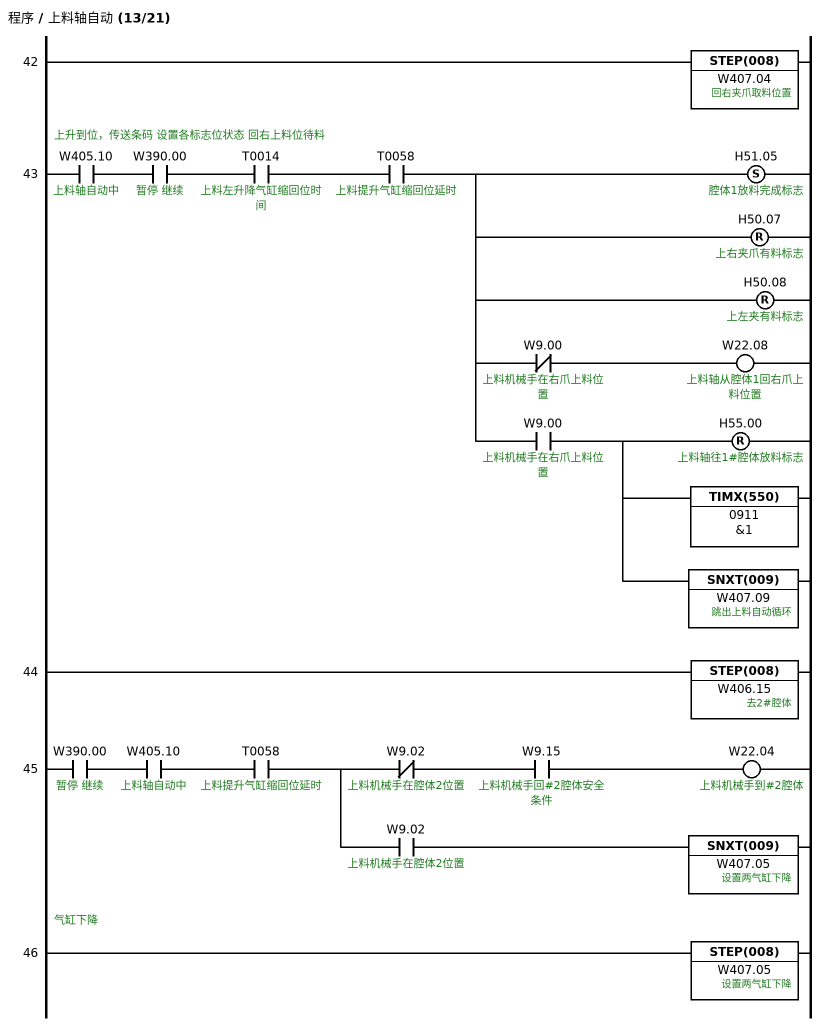
; rung 42
STEP(008) W407.04  ; 回右夹爪取料位置
; rung 43: 上升到位，传送条码 设置各标志位状态 回右上料位待料
LD W405.10  ; 上料轴自动中
AND W390.00  ; 暂停 继续
AND T0014  ; 上料左升降气缸缩回位时间
AND T0058  ; 上料提升气缸缩回位延时
OUT TR0
SET H51.05  ; 腔体1放料完成标志
RSET H50.07  ; 上右夹爪有料标志
RSET H50.08  ; 上左夹有料标志
ANDNOT W9.00  ; 上料机械手在右爪上料位置
OUT W22.08  ; 上料轴从腔体1回右爪上料位置
LD TR0
AND W9.00  ; 上料机械手在右爪上料位置
RSET H55.00  ; 上料轴往1#腔体放料标志
TIMX(550) 0911 &1
SNXT(009) W407.09  ; 跳出上料自动循环
; rung 44
STEP(008) W406.15  ; 去2#腔体
; rung 45
LD W390.00  ; 暂停 继续
AND W405.10  ; 上料轴自动中
AND T0058  ; 上料提升气缸缩回位延时
OUT TR0
ANDNOT W9.02  ; 上料机械手在腔体2位置
AND W9.15  ; 上料机械手回#2腔体安全条件
OUT W22.04  ; 上料机械手到#2腔体
LD TR0
AND W9.02  ; 上料机械手在腔体2位置
SNXT(009) W407.05  ; 设置两气缸下降
; rung 46: 气缸下降
STEP(008) W407.05  ; 设置两气缸下降

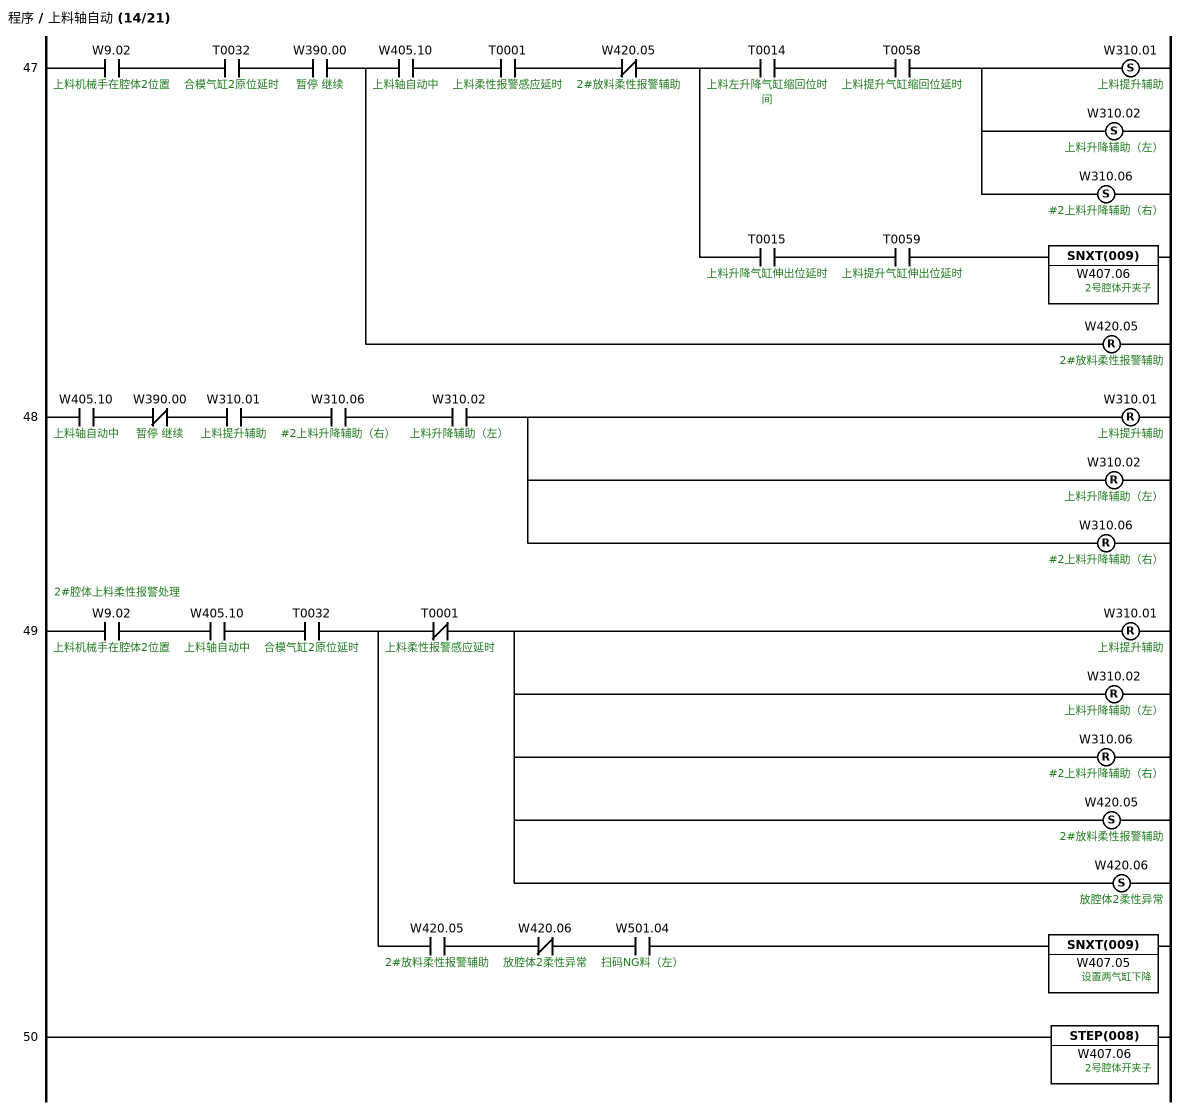
; rung 47
LD W9.02  ; 上料机械手在腔体2位置
AND T0032  ; 合模气缸2原位延时
AND W390.00  ; 暂停 继续
OUT TR0
AND W405.10  ; 上料轴自动中
AND T0001  ; 上料柔性报警感应延时
ANDNOT W420.05  ; 2#放料柔性报警辅助
OUT TR1
AND T0014  ; 上料左升降气缸缩回位时间
AND T0058  ; 上料提升气缸缩回位延时
SET W310.01  ; 上料提升辅助
SET W310.02  ; 上料升降辅助（左）
SET W310.06  ; #2上料升降辅助（右）
LD TR1
AND T0015  ; 上料升降气缸伸出位延时
AND T0059  ; 上料提升气缸伸出位延时
SNXT(009) W407.06  ; 2号腔体开夹子
LD TR0
RSET W420.05  ; 2#放料柔性报警辅助
; rung 48
LD W405.10  ; 上料轴自动中
ANDNOT W390.00  ; 暂停 继续
AND W310.01  ; 上料提升辅助
AND W310.06  ; #2上料升降辅助（右）
AND W310.02  ; 上料升降辅助（左）
RSET W310.01  ; 上料提升辅助
RSET W310.02  ; 上料升降辅助（左）
RSET W310.06  ; #2上料升降辅助（右）
; rung 49: 2#腔体上料柔性报警处理
LD W9.02  ; 上料机械手在腔体2位置
AND W405.10  ; 上料轴自动中
AND T0032  ; 合模气缸2原位延时
OUT TR0
ANDNOT T0001  ; 上料柔性报警感应延时
RSET W310.01  ; 上料提升辅助
RSET W310.02  ; 上料升降辅助（左）
RSET W310.06  ; #2上料升降辅助（右）
SET W420.05  ; 2#放料柔性报警辅助
SET W420.06  ; 放腔体2柔性异常
LD TR0
AND W420.05  ; 2#放料柔性报警辅助
ANDNOT W420.06  ; 放腔体2柔性异常
AND W501.04  ; 扫码NG料（左）
SNXT(009) W407.05  ; 设置两气缸下降
; rung 50
STEP(008) W407.06  ; 2号腔体开夹子

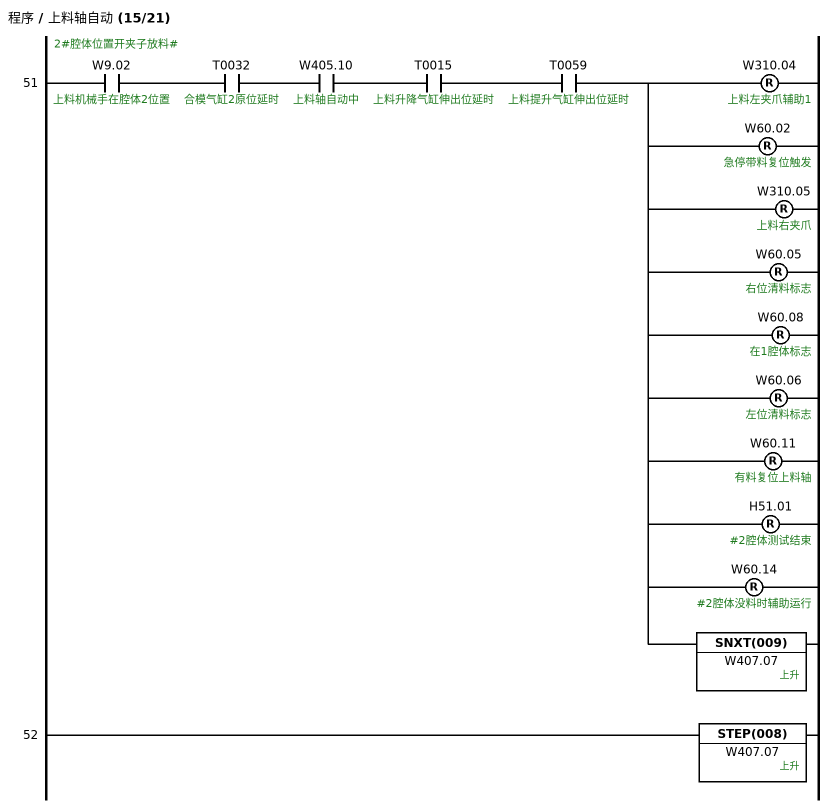
; rung 51: 2#腔体位置开夹子放料#
LD W9.02  ; 上料机械手在腔体2位置
AND T0032  ; 合模气缸2原位延时
AND W405.10  ; 上料轴自动中
AND T0015  ; 上料升降气缸伸出位延时
AND T0059  ; 上料提升气缸伸出位延时
RSET W310.04  ; 上料左夹爪辅助1
RSET W60.02  ; 急停带料复位触发
RSET W310.05  ; 上料右夹爪
RSET W60.05  ; 右位清料标志
RSET W60.08  ; 在1腔体标志
RSET W60.06  ; 左位清料标志
RSET W60.11  ; 有料复位上料轴
RSET H51.01  ; #2腔体测试结束
RSET W60.14  ; #2腔体没料时辅助运行
SNXT(009) W407.07  ; 上升
; rung 52
STEP(008) W407.07  ; 上升

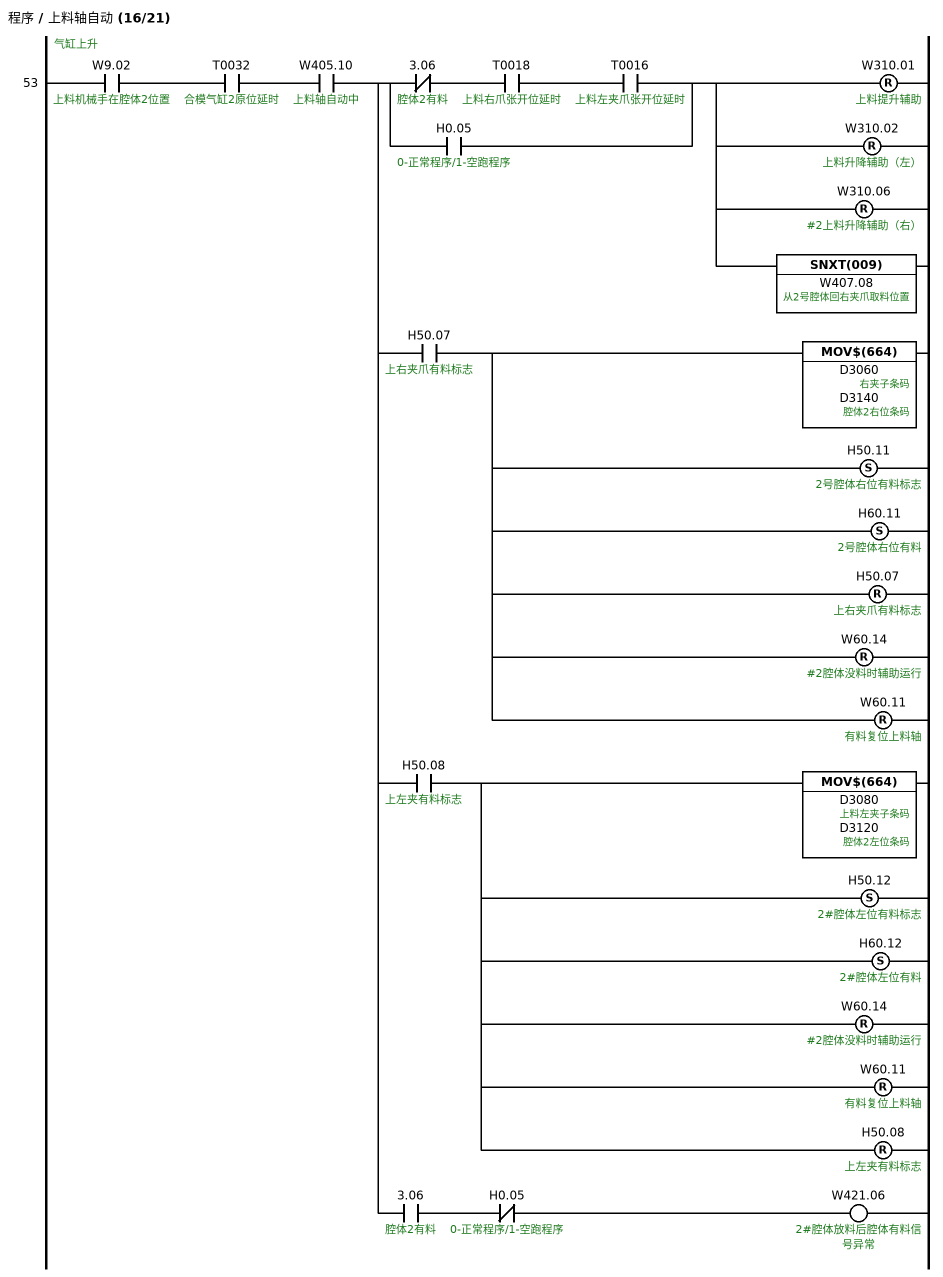
; rung 53: 气缸上升
LD W9.02  ; 上料机械手在腔体2位置
AND T0032  ; 合模气缸2原位延时
AND W405.10  ; 上料轴自动中
OUT TR0
LDNOT 3.06  ; 腔体2有料
AND T0018  ; 上料右爪张开位延时
AND T0016  ; 上料左夹爪张开位延时
OR H0.05  ; 0-正常程序/1-空跑程序
ANDLD
RSET W310.01  ; 上料提升辅助
RSET W310.02  ; 上料升降辅助（左）
RSET W310.06  ; #2上料升降辅助（右）
SNXT(009) W407.08  ; 从2号腔体回右夹爪取料位置
LD TR0
AND H50.07  ; 上右夹爪有料标志
MOV$(664) D3060 D3140  ; 右夹子条码, 腔体2右位条码
SET H50.11  ; 2号腔体右位有料标志
SET H60.11  ; 2号腔体右位有料
RSET H50.07  ; 上右夹爪有料标志
RSET W60.14  ; #2腔体没料时辅助运行
RSET W60.11  ; 有料复位上料轴
LD TR0
AND H50.08  ; 上左夹有料标志
MOV$(664) D3080 D3120  ; 上料左夹子条码, 腔体2左位条码
SET H50.12  ; 2#腔体左位有料标志
SET H60.12  ; 2#腔体左位有料
RSET W60.14  ; #2腔体没料时辅助运行
RSET W60.11  ; 有料复位上料轴
RSET H50.08  ; 上左夹有料标志
LD TR0
AND 3.06  ; 腔体2有料
ANDNOT H0.05  ; 0-正常程序/1-空跑程序
OUT W421.06  ; 2#腔体放料后腔体有料信号异常

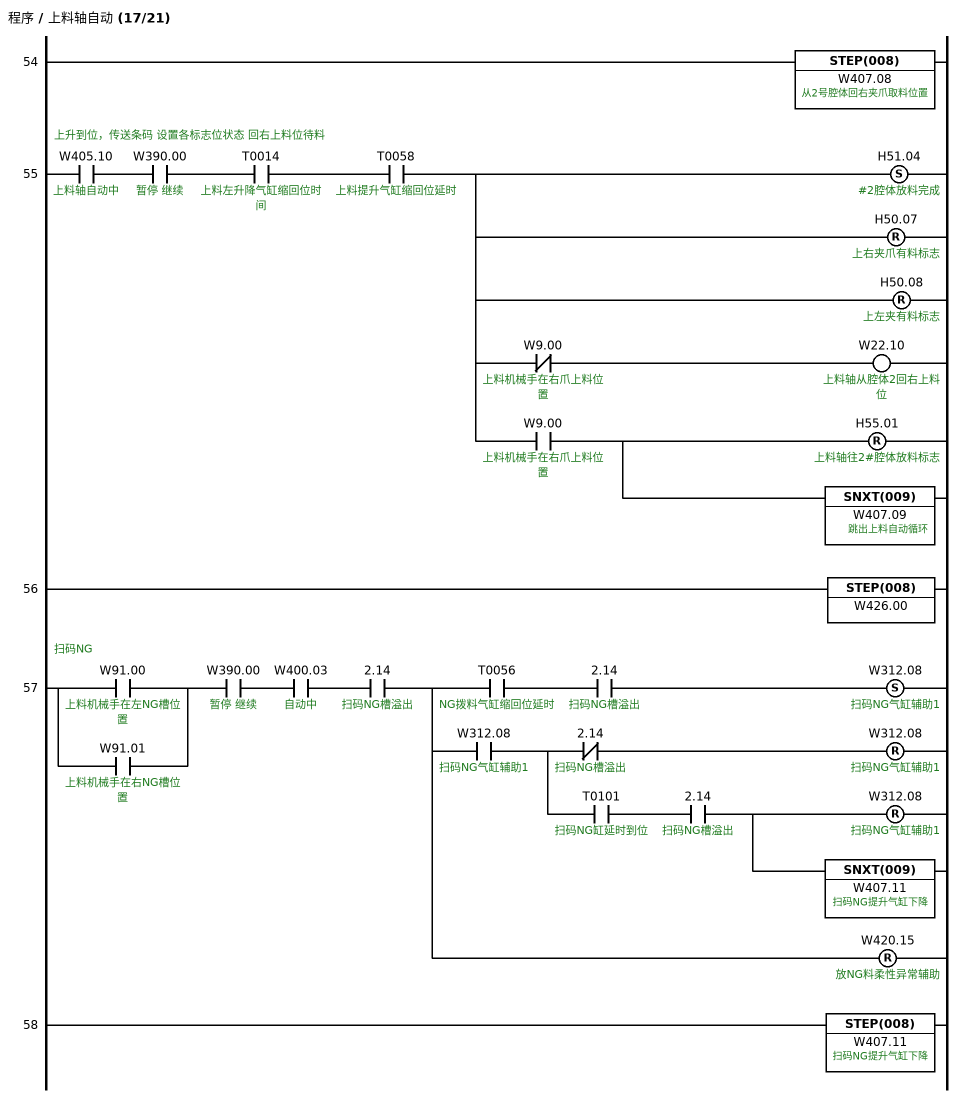
; rung 54
STEP(008) W407.08  ; 从2号腔体回右夹爪取料位置
; rung 55: 上升到位，传送条码 设置各标志位状态 回右上料位待料
LD W405.10  ; 上料轴自动中
AND W390.00  ; 暂停 继续
AND T0014  ; 上料左升降气缸缩回位时间
AND T0058  ; 上料提升气缸缩回位延时
OUT TR0
SET H51.04  ; #2腔体放料完成
RSET H50.07  ; 上右夹爪有料标志
RSET H50.08  ; 上左夹有料标志
ANDNOT W9.00  ; 上料机械手在右爪上料位置
OUT W22.10  ; 上料轴从腔体2回右上料位
LD TR0
AND W9.00  ; 上料机械手在右爪上料位置
RSET H55.01  ; 上料轴往2#腔体放料标志
SNXT(009) W407.09  ; 跳出上料自动循环
; rung 56
STEP(008) W426.00
; rung 57: 扫码NG
LD W91.00  ; 上料机械手在左NG槽位置
OR W91.01  ; 上料机械手在右NG槽位置
AND W390.00  ; 暂停 继续
AND W400.03  ; 自动中
AND 2.14  ; 扫码NG槽溢出
OUT TR0
AND T0056  ; NG拨料气缸缩回位延时
AND 2.14  ; 扫码NG槽溢出
SET W312.08  ; 扫码NG气缸辅助1
LD TR0
AND W312.08  ; 扫码NG气缸辅助1
OUT TR1
ANDNOT 2.14  ; 扫码NG槽溢出
RSET W312.08  ; 扫码NG气缸辅助1
LD TR1
AND T0101  ; 扫码NG缸延时到位
AND 2.14  ; 扫码NG槽溢出
RSET W312.08  ; 扫码NG气缸辅助1
SNXT(009) W407.11  ; 扫码NG提升气缸下降
LD TR0
RSET W420.15  ; 放NG料柔性异常辅助
; rung 58
STEP(008) W407.11  ; 扫码NG提升气缸下降

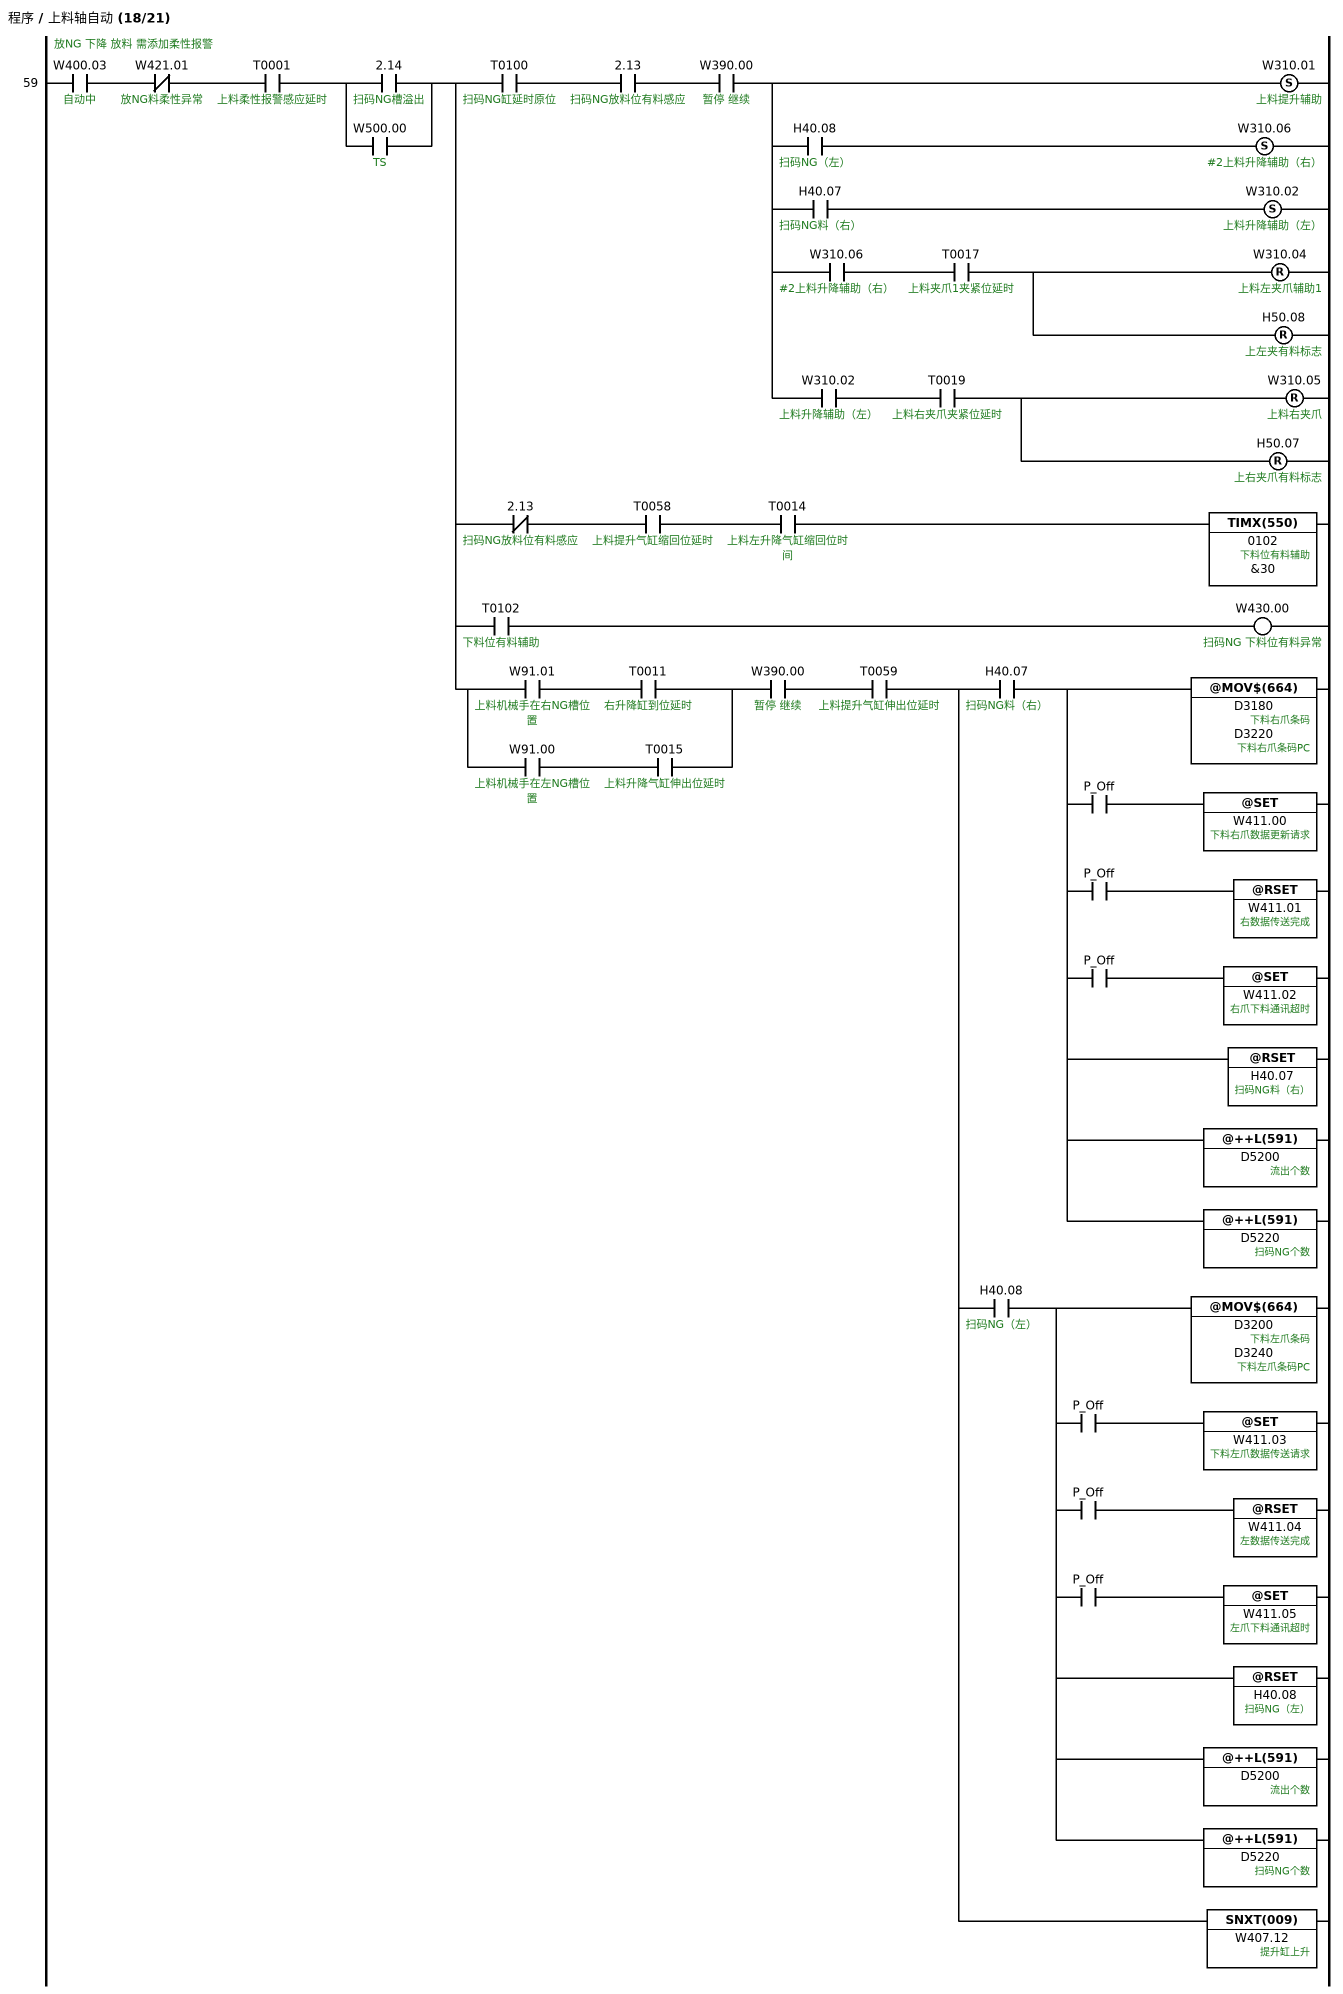
; rung 59: 放NG 下降 放料 需添加柔性报警
LD W400.03  ; 自动中
ANDNOT W421.01  ; 放NG料柔性异常
AND T0001  ; 上料柔性报警感应延时
LD 2.14  ; 扫码NG槽溢出
OR W500.00  ; TS
ANDLD
OUT TR0
AND T0100  ; 扫码NG缸延时原位
AND 2.13  ; 扫码NG放料位有料感应
AND W390.00  ; 暂停 继续
OUT TR1
SET W310.01  ; 上料提升辅助
AND H40.08  ; 扫码NG（左）
SET W310.06  ; #2上料升降辅助（右）
LD TR1
AND H40.07  ; 扫码NG料（右）
SET W310.02  ; 上料升降辅助（左）
LD TR1
AND W310.06  ; #2上料升降辅助（右）
AND T0017  ; 上料夹爪1夹紧位延时
RSET W310.04  ; 上料左夹爪辅助1
RSET H50.08  ; 上左夹有料标志
LD TR1
AND W310.02  ; 上料升降辅助（左）
AND T0019  ; 上料右夹爪夹紧位延时
RSET W310.05  ; 上料右夹爪
RSET H50.07  ; 上右夹爪有料标志
LD TR0
ANDNOT 2.13  ; 扫码NG放料位有料感应
AND T0058  ; 上料提升气缸缩回位延时
AND T0014  ; 上料左升降气缸缩回位时间
TIMX(550) 0102 &30  ; 下料位有料辅助
LD TR0
AND T0102  ; 下料位有料辅助
OUT W430.00  ; 扫码NG 下料位有料异常
LD TR0
LD W91.01  ; 上料机械手在右NG槽位置
AND T0011  ; 右升降缸到位延时
LD W91.00  ; 上料机械手在左NG槽位置
AND T0015  ; 上料升降气缸伸出位延时
ORLD
ANDLD
AND W390.00  ; 暂停 继续
AND T0059  ; 上料提升气缸伸出位延时
OUT TR0
AND H40.07  ; 扫码NG料（右）
OUT TR1
@MOV$(664) D3180 D3220  ; 下料右爪条码, 下料右爪条码PC
AND P_Off
@SET W411.00  ; 下料右爪数据更新请求
LD TR1
AND P_Off
@RSET W411.01  ; 右数据传送完成
LD TR1
AND P_Off
@SET W411.02  ; 右爪下料通讯超时
LD TR1
@RSET H40.07  ; 扫码NG料（右）
@++L(591) D5200  ; 流出个数
@++L(591) D5220  ; 扫码NG个数
LD TR0
AND H40.08  ; 扫码NG（左）
OUT TR1
@MOV$(664) D3200 D3240  ; 下料左爪条码, 下料左爪条码PC
AND P_Off
@SET W411.03  ; 下料左爪数据传送请求
LD TR1
AND P_Off
@RSET W411.04  ; 左数据传送完成
LD TR1
AND P_Off
@SET W411.05  ; 左爪下料通讯超时
LD TR1
@RSET H40.08  ; 扫码NG（左）
@++L(591) D5200  ; 流出个数
@++L(591) D5220  ; 扫码NG个数
LD TR0
SNXT(009) W407.12  ; 提升缸上升

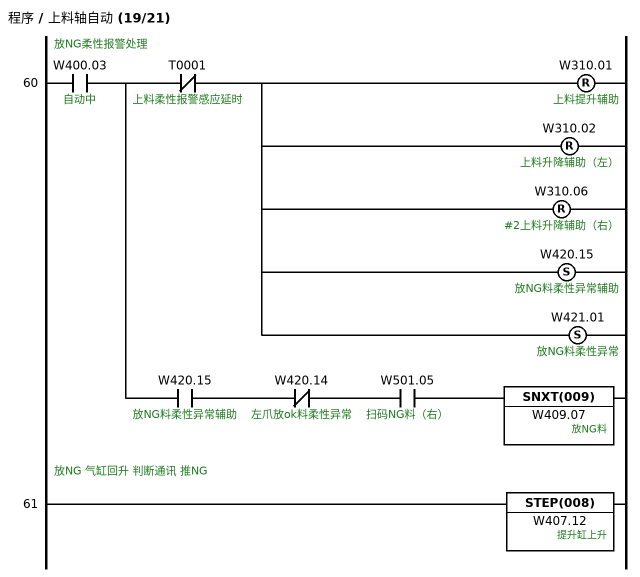
; rung 60: 放NG柔性报警处理
LD W400.03  ; 自动中
OUT TR0
ANDNOT T0001  ; 上料柔性报警感应延时
RSET W310.01  ; 上料提升辅助
RSET W310.02  ; 上料升降辅助（左）
RSET W310.06  ; #2上料升降辅助（右）
SET W420.15  ; 放NG料柔性异常辅助
SET W421.01  ; 放NG料柔性异常
LD TR0
AND W420.15  ; 放NG料柔性异常辅助
ANDNOT W420.14  ; 左爪放ok料柔性异常
AND W501.05  ; 扫码NG料（右）
SNXT(009) W409.07  ; 放NG料
; rung 61: 放NG 气缸回升 判断通讯 推NG
STEP(008) W407.12  ; 提升缸上升

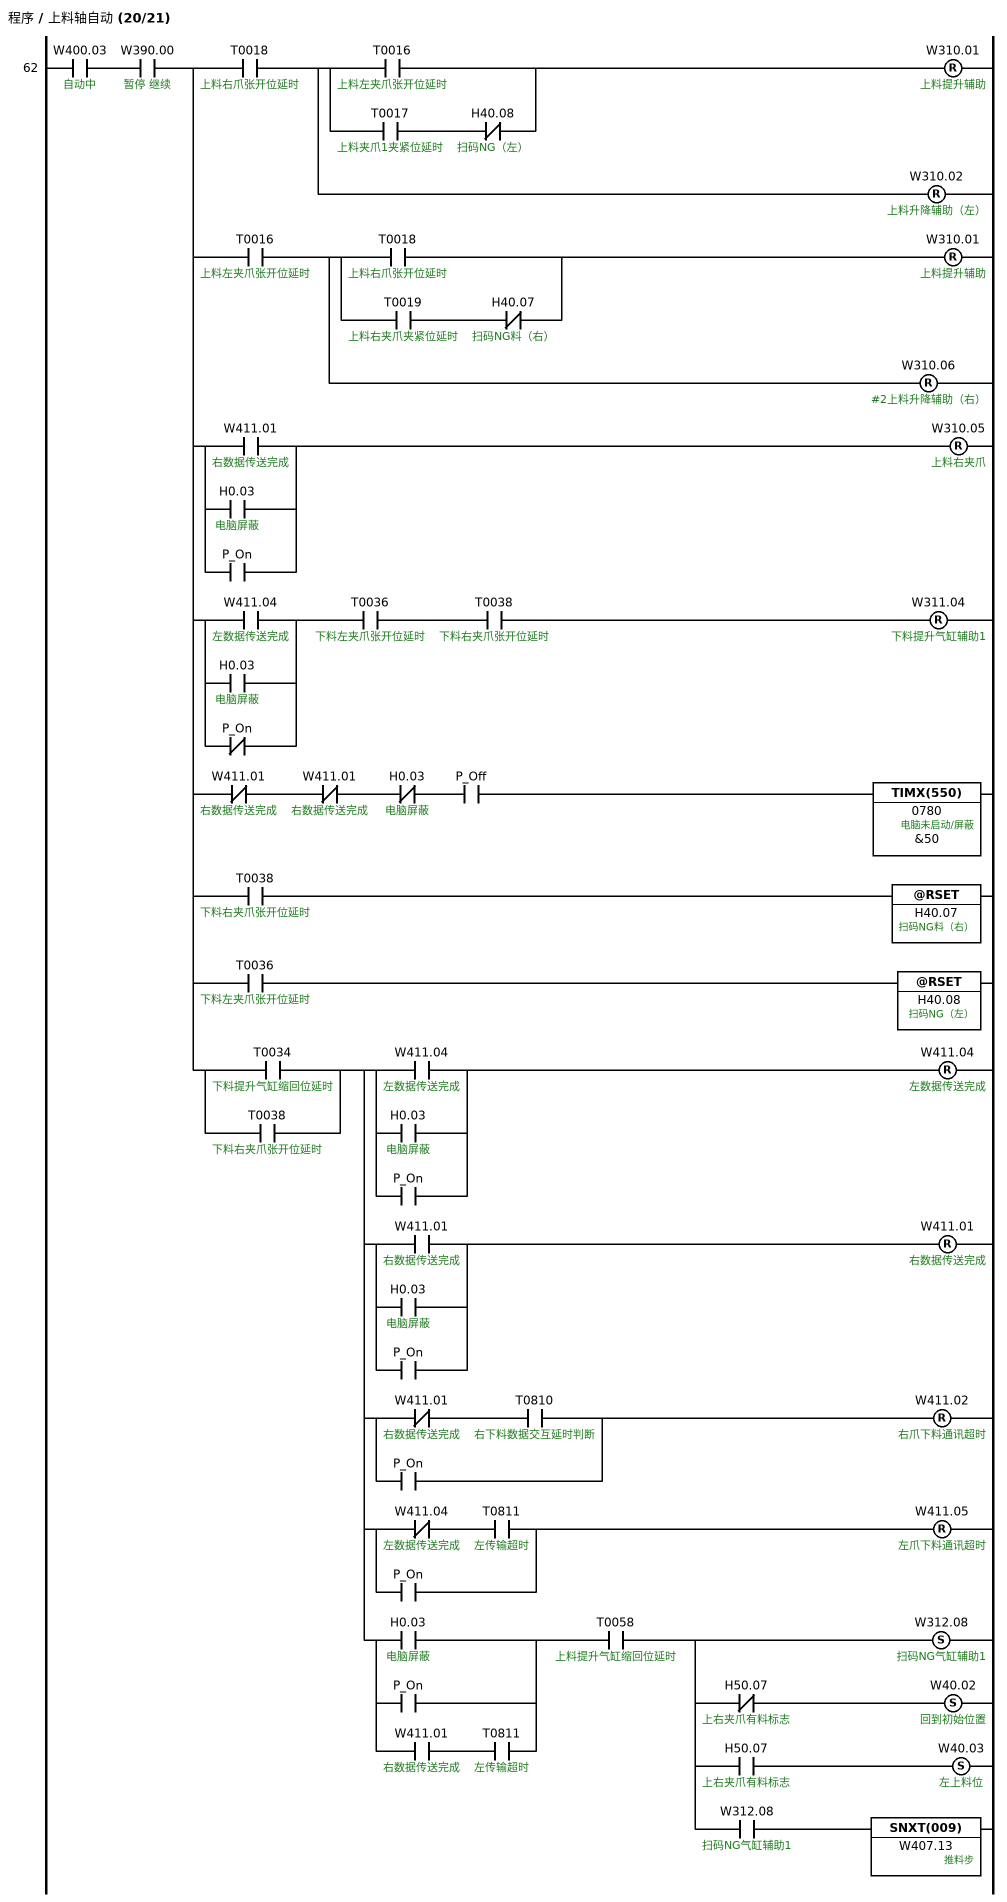
; rung 62
LD W400.03  ; 自动中
AND W390.00  ; 暂停 继续
OUT TR0
AND T0018  ; 上料右爪张开位延时
OUT TR1
LD T0016  ; 上料左夹爪张开位延时
LD T0017  ; 上料夹爪1夹紧位延时
ANDNOT H40.08  ; 扫码NG（左）
ORLD
ANDLD
RSET W310.01  ; 上料提升辅助
LD TR1
RSET W310.02  ; 上料升降辅助（左）
LD TR0
AND T0016  ; 上料左夹爪张开位延时
OUT TR1
LD T0018  ; 上料右爪张开位延时
LD T0019  ; 上料右夹爪夹紧位延时
ANDNOT H40.07  ; 扫码NG料（右）
ORLD
ANDLD
RSET W310.01  ; 上料提升辅助
LD TR1
RSET W310.06  ; #2上料升降辅助（右）
LD TR0
LD W411.01  ; 右数据传送完成
OR H0.03  ; 电脑屏蔽
OR P_On
ANDLD
RSET W310.05  ; 上料右夹爪
LD TR0
LD W411.04  ; 左数据传送完成
OR H0.03  ; 电脑屏蔽
ORNOT P_On
ANDLD
AND T0036  ; 下料左夹爪张开位延时
AND T0038  ; 下料右夹爪张开位延时
RSET W311.04  ; 下料提升气缸辅助1
LD TR0
ANDNOT W411.01  ; 右数据传送完成
ANDNOT W411.01  ; 右数据传送完成
ANDNOT H0.03  ; 电脑屏蔽
AND P_Off
TIMX(550) 0780 &50  ; 电脑未启动/屏蔽
LD TR0
AND T0038  ; 下料右夹爪张开位延时
@RSET H40.07  ; 扫码NG料（右）
LD TR0
AND T0036  ; 下料左夹爪张开位延时
@RSET H40.08  ; 扫码NG（左）
LD TR0
LD T0034  ; 下料提升气缸缩回位延时
OR T0038  ; 下料右夹爪张开位延时
ANDLD
OUT TR0
LD W411.04  ; 左数据传送完成
OR H0.03  ; 电脑屏蔽
OR P_On
ANDLD
RSET W411.04  ; 左数据传送完成
LD TR0
LD W411.01  ; 右数据传送完成
OR H0.03  ; 电脑屏蔽
OR P_On
ANDLD
RSET W411.01  ; 右数据传送完成
LD TR0
LDNOT W411.01  ; 右数据传送完成
AND T0810  ; 右下料数据交互延时判断
OR P_On
ANDLD
RSET W411.02  ; 右爪下料通讯超时
LD TR0
LDNOT W411.04  ; 左数据传送完成
AND T0811  ; 左传输超时
OR P_On
ANDLD
RSET W411.05  ; 左爪下料通讯超时
LD TR0
LD H0.03  ; 电脑屏蔽
OR P_On
LD W411.01  ; 右数据传送完成
AND T0811  ; 左传输超时
ORLD
ANDLD
AND T0058  ; 上料提升气缸缩回位延时
OUT TR0
SET W312.08  ; 扫码NG气缸辅助1
ANDNOT H50.07  ; 上右夹爪有料标志
SET W40.02  ; 回到初始位置
LD TR0
AND H50.07  ; 上右夹爪有料标志
SET W40.03  ; 左上料位
LD TR0
AND W312.08  ; 扫码NG气缸辅助1
SNXT(009) W407.13  ; 推料步

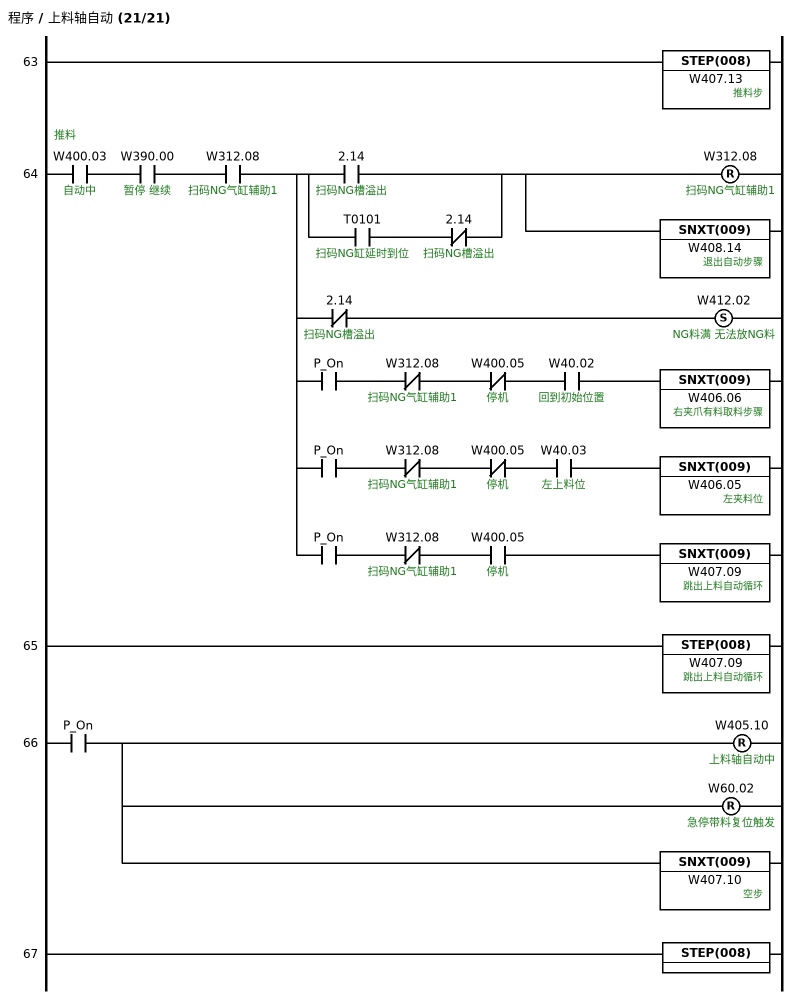
; rung 63
STEP(008) W407.13  ; 推料步
; rung 64: 推料
LD W400.03  ; 自动中
AND W390.00  ; 暂停 继续
AND W312.08  ; 扫码NG气缸辅助1
OUT TR0
LD 2.14  ; 扫码NG槽溢出
LD T0101  ; 扫码NG缸延时到位
ANDNOT 2.14  ; 扫码NG槽溢出
ORLD
ANDLD
RSET W312.08  ; 扫码NG气缸辅助1
SNXT(009) W408.14  ; 退出自动步骤
LD TR0
ANDNOT 2.14  ; 扫码NG槽溢出
SET W412.02  ; NG料满 无法放NG料
LD TR0
AND P_On
ANDNOT W312.08  ; 扫码NG气缸辅助1
ANDNOT W400.05  ; 停机
AND W40.02  ; 回到初始位置
SNXT(009) W406.06  ; 右夹爪有料取料步骤
LD TR0
AND P_On
ANDNOT W312.08  ; 扫码NG气缸辅助1
ANDNOT W400.05  ; 停机
AND W40.03  ; 左上料位
SNXT(009) W406.05  ; 左夹料位
LD TR0
AND P_On
ANDNOT W312.08  ; 扫码NG气缸辅助1
AND W400.05  ; 停机
SNXT(009) W407.09  ; 跳出上料自动循环
; rung 65
STEP(008) W407.09  ; 跳出上料自动循环
; rung 66
LD P_On
RSET W405.10  ; 上料轴自动中
RSET W60.02  ; 急停带料复位触发
SNXT(009) W407.10  ; 空步
; rung 67
STEP(008)

### Section 腔体1自动

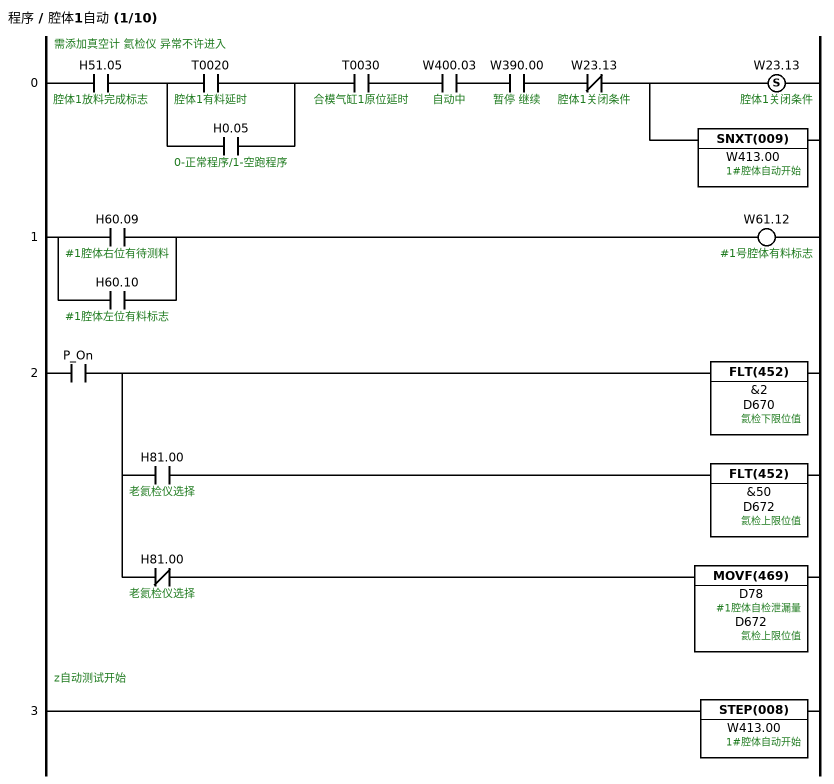
; rung 0: 需添加真空计 氦检仪 异常不许进入
LD H51.05  ; 腔体1放料完成标志
LD T0020  ; 腔体1有料延时
OR H0.05  ; 0-正常程序/1-空跑程序
ANDLD
AND T0030  ; 合模气缸1原位延时
AND W400.03  ; 自动中
AND W390.00  ; 暂停 继续
ANDNOT W23.13  ; 腔体1关闭条件
SET W23.13  ; 腔体1关闭条件
SNXT(009) W413.00  ; 1#腔体自动开始
; rung 1
LD H60.09  ; #1腔体右位有待测料
OR H60.10  ; #1腔体左位有料标志
OUT W61.12  ; #1号腔体有料标志
; rung 2
LD P_On
OUT TR0
FLT(452) &2 D670  ; 氦检下限位值
AND H81.00  ; 老氦检仪选择
FLT(452) &50 D672  ; 氦检上限位值
LD TR0
ANDNOT H81.00  ; 老氦检仪选择
MOVF(469) D78 D672  ; #1腔体自检泄漏量, 氦检上限位值
; rung 3: z自动测试开始
STEP(008) W413.00  ; 1#腔体自动开始

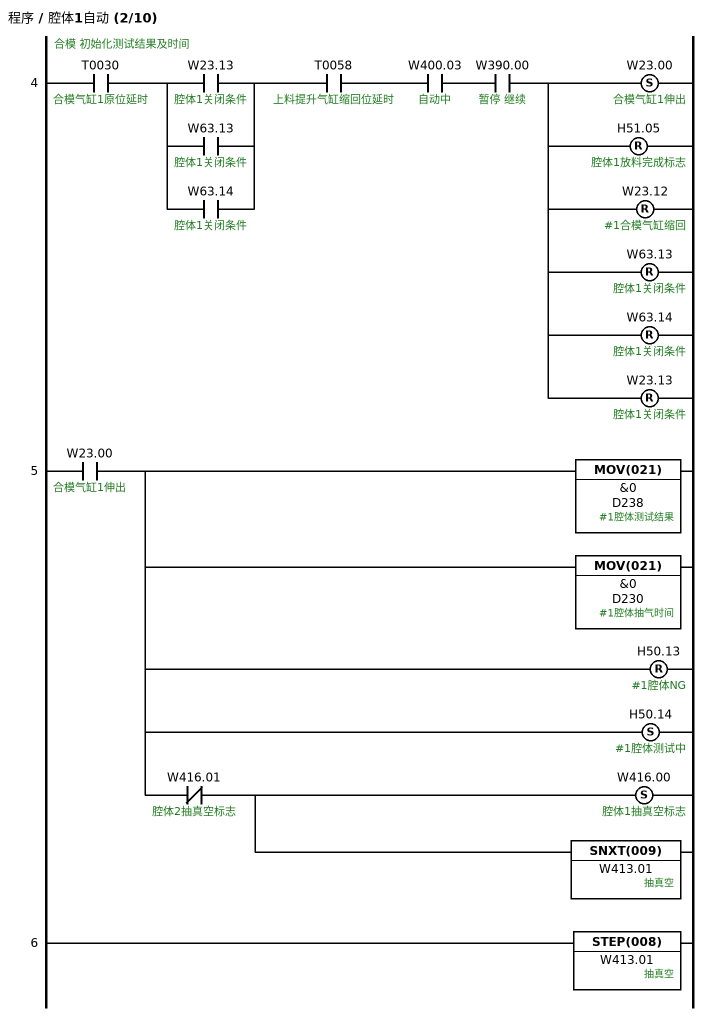
; rung 4: 合模 初始化测试结果及时间
LD T0030  ; 合模气缸1原位延时
LD W23.13  ; 腔体1关闭条件
OR W63.13  ; 腔体1关闭条件
OR W63.14  ; 腔体1关闭条件
ANDLD
AND T0058  ; 上料提升气缸缩回位延时
AND W400.03  ; 自动中
AND W390.00  ; 暂停 继续
SET W23.00  ; 合模气缸1伸出
RSET H51.05  ; 腔体1放料完成标志
RSET W23.12  ; #1合模气缸缩回
RSET W63.13  ; 腔体1关闭条件
RSET W63.14  ; 腔体1关闭条件
RSET W23.13  ; 腔体1关闭条件
; rung 5
LD W23.00  ; 合模气缸1伸出
MOV(021) &0 D238  ; #1腔体测试结果
MOV(021) &0 D230  ; #1腔体抽气时间
RSET H50.13  ; #1腔体NG
SET H50.14  ; #1腔体测试中
ANDNOT W416.01  ; 腔体2抽真空标志
SET W416.00  ; 腔体1抽真空标志
SNXT(009) W413.01  ; 抽真空
; rung 6
STEP(008) W413.01  ; 抽真空

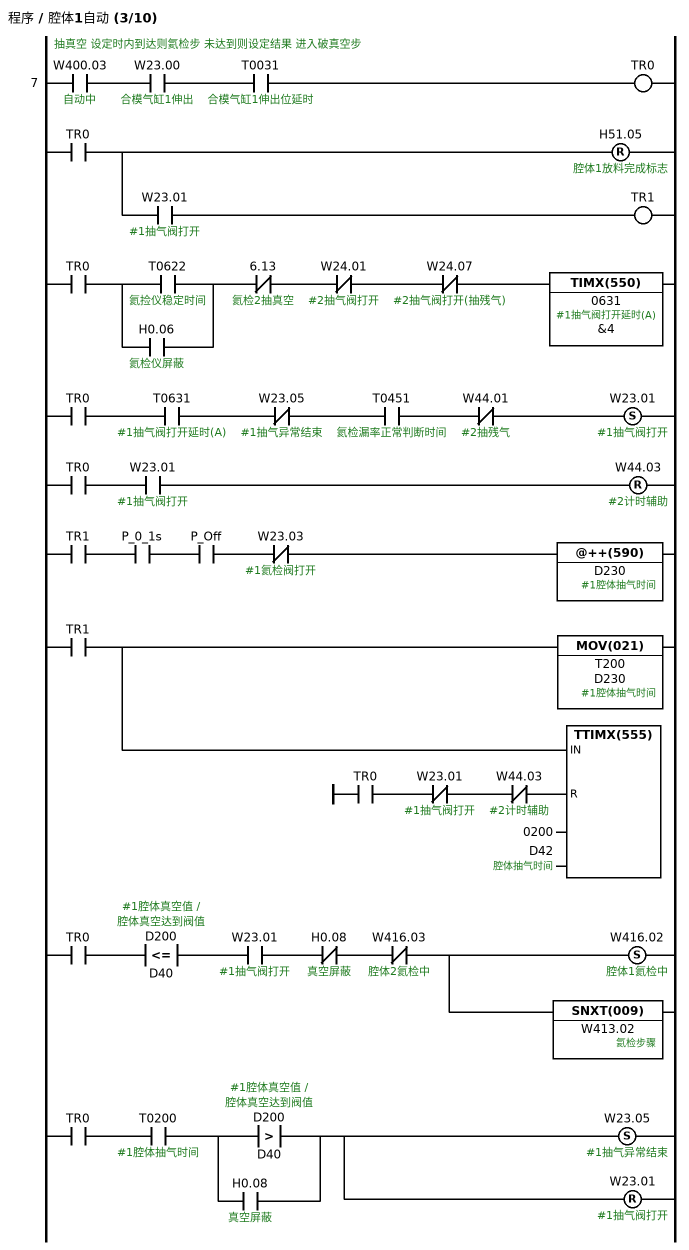
; rung 7: 抽真空 设定时内到达则氦检步 未达到则设定结果 进入破真空步
LD W400.03  ; 自动中
AND W23.00  ; 合模气缸1伸出
AND T0031  ; 合模气缸1伸出位延时
OUT TR0
LD T0622  ; 氦捡仪稳定时间
OR H0.06  ; 氦检仪屏蔽
ANDLD
ANDNOT 6.13  ; 氦检2抽真空
ANDNOT W24.01  ; #2抽气阀打开
ANDNOT W24.07  ; #2抽气阀打开(抽残气)
TIMX(550) 0631 &4  ; #1抽气阀打开延时(A)
LD TR0
AND T0631  ; #1抽气阀打开延时(A)
ANDNOT W23.05  ; #1抽气异常结束
AND T0451  ; 氦检漏率正常判断时间
ANDNOT W44.01  ; #2抽残气
SET W23.01  ; #1抽气阀打开
LD TR0
AND W23.01  ; #1抽气阀打开
RSET W44.03  ; #2计时辅助
LD TR0
RSET H51.05  ; 腔体1放料完成标志
AND W23.01  ; #1抽气阀打开
OUT TR1
AND P_0_1s
AND P_Off
ANDNOT W23.03  ; #1氦检阀打开
@++(590) D230  ; #1腔体抽气时间
LD TR1
MOV(021) T200 D230  ; #1腔体抽气时间
LD TR0
ANDNOT W23.01  ; #1抽气阀打开
ANDNOT W44.03  ; #2计时辅助
TTIMX(555) 0200 D42  ; 腔体抽气时间, #1腔体抽气时间
LD TR0
AND<=F(332) D200 D40  ; #1腔体真空值, 腔体真空达到阀值
AND W23.01  ; #1抽气阀打开
ANDNOT H0.08  ; 真空屏蔽
ANDNOT W416.03  ; 腔体2氦检中
SET W416.02  ; 腔体1氦检中
SNXT(009) W413.02  ; 氦检步骤
LD TR0
AND T0200  ; #1腔体抽气时间
LD>F(333) D200 D40  ; #1腔体真空值, 腔体真空达到阀值
OR H0.08  ; 真空屏蔽
ANDLD
SET W23.05  ; #1抽气异常结束
RSET W23.01  ; #1抽气阀打开

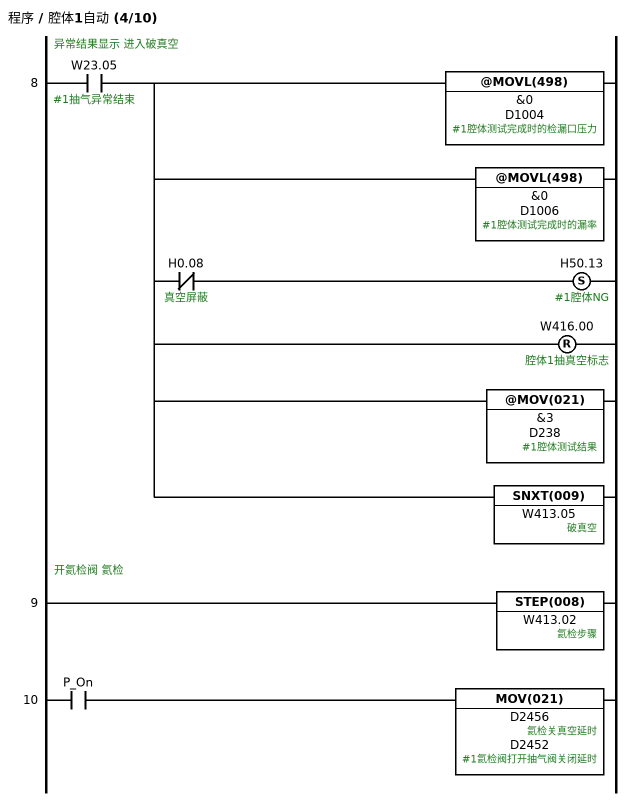
; rung 8: 异常结果显示 进入破真空
LD W23.05  ; #1抽气异常结束
OUT TR0
@MOVL(498) &0 D1004  ; #1腔体测试完成时的检漏口压力
@MOVL(498) &0 D1006  ; #1腔体测试完成时的漏率
ANDNOT H0.08  ; 真空屏蔽
SET H50.13  ; #1腔体NG
LD TR0
RSET W416.00  ; 腔体1抽真空标志
@MOV(021) &3 D238  ; #1腔体测试结果
SNXT(009) W413.05  ; 破真空
; rung 9: 开氦检阀 氦检
STEP(008) W413.02  ; 氦检步骤
; rung 10
LD P_On
MOV(021) D2456 D2452  ; 氦检关真空延时, #1氦检阀打开抽气阀关闭延时

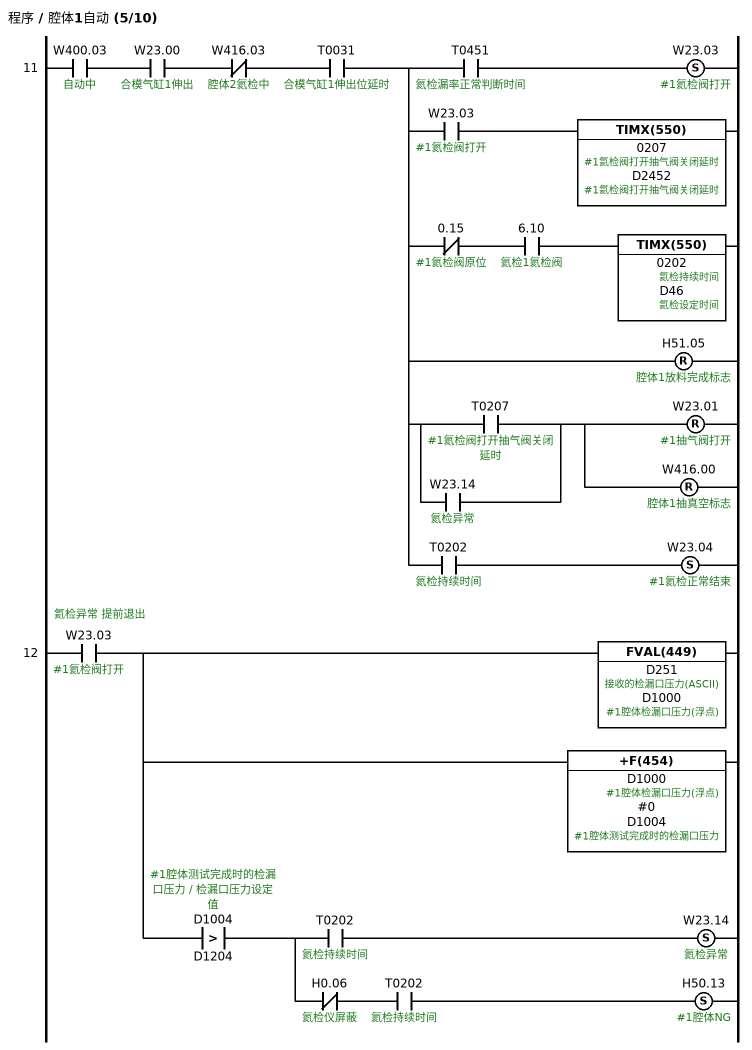
; rung 11
LD W400.03  ; 自动中
AND W23.00  ; 合模气缸1伸出
ANDNOT W416.03  ; 腔体2氦检中
AND T0031  ; 合模气缸1伸出位延时
OUT TR0
AND T0451  ; 氦检漏率正常判断时间
SET W23.03  ; #1氦检阀打开
LD TR0
AND W23.03  ; #1氦检阀打开
TIMX(550) 0207 D2452  ; #1氦检阀打开抽气阀关闭延时
LD TR0
ANDNOT 0.15  ; #1氦检阀原位
AND 6.10  ; 氦检1氦检阀
TIMX(550) 0202 D46  ; 氦检设定时间, 氦检持续时间
LD TR0
RSET H51.05  ; 腔体1放料完成标志
LD T0207  ; #1氦检阀打开抽气阀关闭延时
OR W23.14  ; 氦检异常
ANDLD
RSET W23.01  ; #1抽气阀打开
RSET W416.00  ; 腔体1抽真空标志
LD TR0
AND T0202  ; 氦检持续时间
SET W23.04  ; #1氦检正常结束
; rung 12: 氦检异常 提前退出
LD W23.03  ; #1氦检阀打开
FVAL(449) D251 D1000  ; 接收的检漏口压力(ASCII), #1腔体检漏口压力(浮点)
+F(454) D1000 #0 D1004  ; #1腔体检漏口压力(浮点), #1腔体测试完成时的检漏口压力
AND>F(333) D1004 D1204  ; #1腔体测试完成时的检漏口压力, 检漏口压力设定值
OUT TR0
AND T0202  ; 氦检持续时间
SET W23.14  ; 氦检异常
LD TR0
ANDNOT H0.06  ; 氦检仪屏蔽
AND T0202  ; 氦检持续时间
SET H50.13  ; #1腔体NG

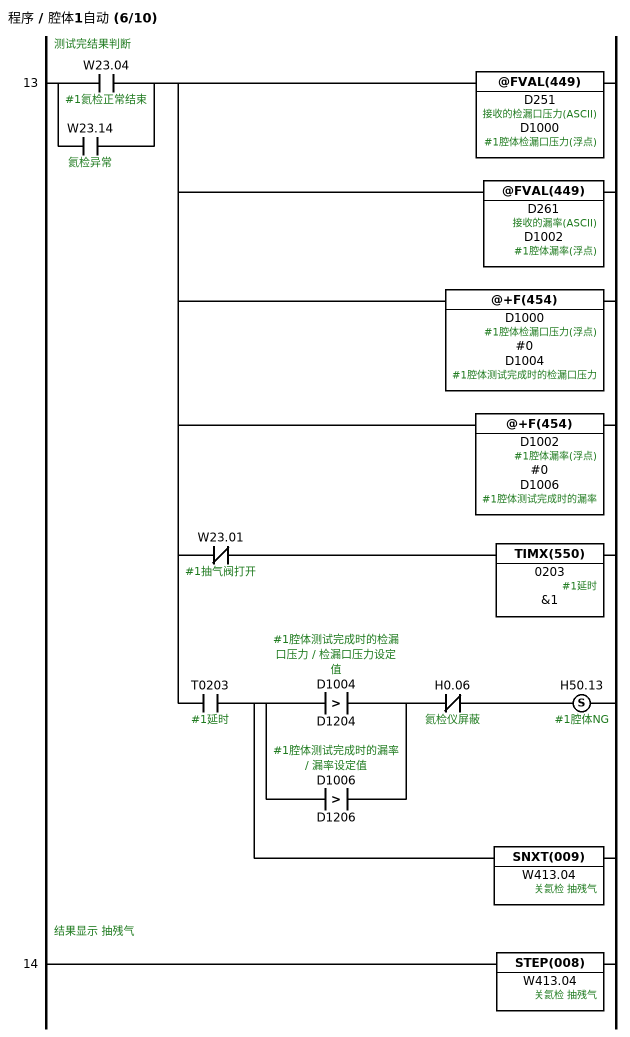
; rung 13: 测试完结果判断
LD W23.04  ; #1氦检正常结束
OR W23.14  ; 氦检异常
OUT TR0
@FVAL(449) D251 D1000  ; 接收的检漏口压力(ASCII), #1腔体检漏口压力(浮点)
@FVAL(449) D261 D1002  ; 接收的漏率(ASCII), #1腔体漏率(浮点)
@+F(454) D1000 #0 D1004  ; #1腔体检漏口压力(浮点), #1腔体测试完成时的检漏口压力
@+F(454) D1002 #0 D1006  ; #1腔体漏率(浮点), #1腔体测试完成时的漏率
ANDNOT W23.01  ; #1抽气阀打开
TIMX(550) 0203 &1  ; #1延时
LD TR0
AND T0203  ; #1延时
OUT TR0
LD>F(333) D1004 D1204  ; #1腔体测试完成时的检漏口压力, 检漏口压力设定值
OR>F(333) D1006 D1206  ; #1腔体测试完成时的漏率, 漏率设定值
ANDLD
ANDNOT H0.06  ; 氦检仪屏蔽
SET H50.13  ; #1腔体NG
LD TR0
SNXT(009) W413.04  ; 关氦检 抽残气
; rung 14: 结果显示 抽残气
STEP(008) W413.04  ; 关氦检 抽残气

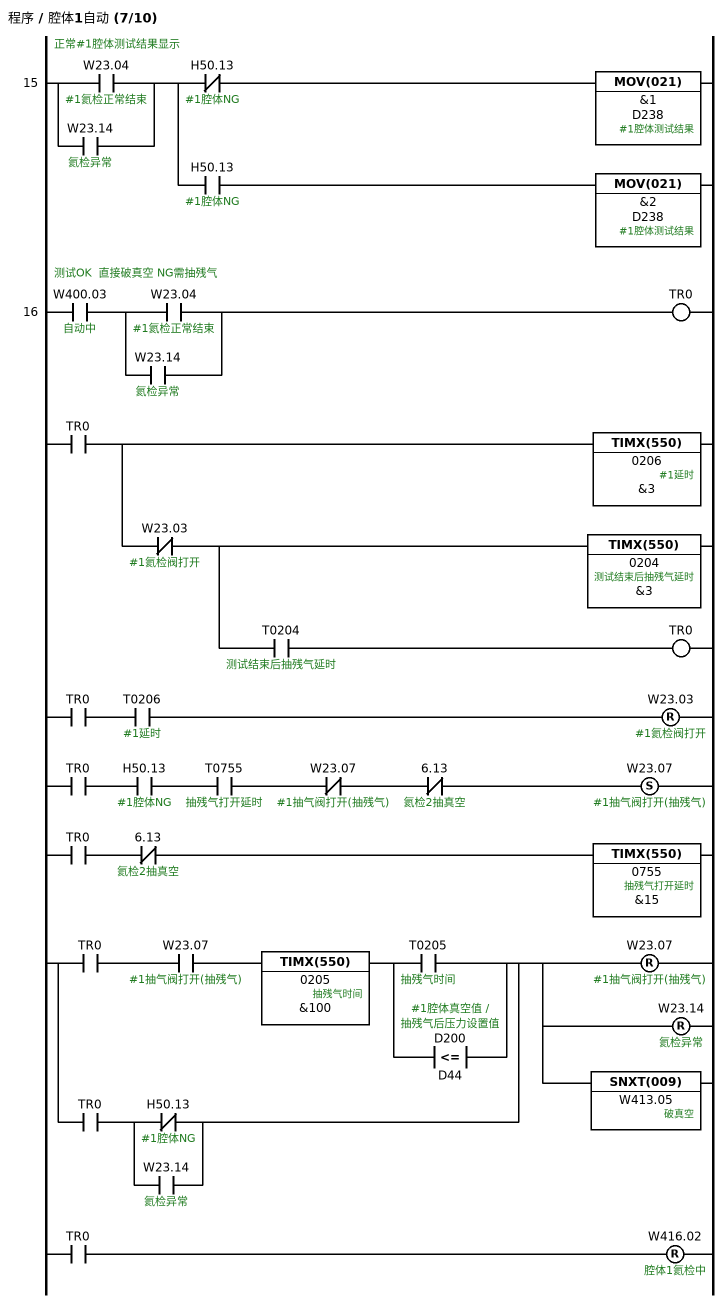
; rung 15: 正常#1腔体测试结果显示
LD W23.04  ; #1氦检正常结束
OR W23.14  ; 氦检异常
OUT TR0
ANDNOT H50.13  ; #1腔体NG
MOV(021) &1 D238  ; #1腔体测试结果
LD TR0
AND H50.13  ; #1腔体NG
MOV(021) &2 D238  ; #1腔体测试结果
; rung 16: 测试OK  直接破真空 NG需抽残气
LD W400.03  ; 自动中
LD W23.04  ; #1氦检正常结束
OR W23.14  ; 氦检异常
ANDLD
OUT TR0
AND T0206  ; #1延时
RSET W23.03  ; #1氦检阀打开
LD TR0
TIMX(550) 0206 &3  ; #1延时
ANDNOT W23.03  ; #1氦检阀打开
TIMX(550) 0204 &3  ; 测试结束后抽残气延时
AND T0204  ; 测试结束后抽残气延时
OUT TR0
AND H50.13  ; #1腔体NG
AND T0755  ; 抽残气打开延时
ANDNOT W23.07  ; #1抽气阀打开(抽残气)
ANDNOT 6.13  ; 氦检2抽真空
SET W23.07  ; #1抽气阀打开(抽残气)
LD TR0
ANDNOT 6.13  ; 氦检2抽真空
TIMX(550) 0755 &15  ; 抽残气打开延时
LD TR0
AND W23.07  ; #1抽气阀打开(抽残气)
TIMX(550) 0205 &100  ; 抽残气时间
LD T0205  ; 抽残气时间
OR<=F(332) D200 D44  ; #1腔体真空值, 抽残气后压力设置值
ANDLD
LD TR0
LDNOT H50.13  ; #1腔体NG
OR W23.14  ; 氦检异常
ANDLD
ORLD
RSET W23.07  ; #1抽气阀打开(抽残气)
RSET W23.14  ; 氦检异常
SNXT(009) W413.05  ; 破真空
LD TR0
RSET W416.02  ; 腔体1氦检中

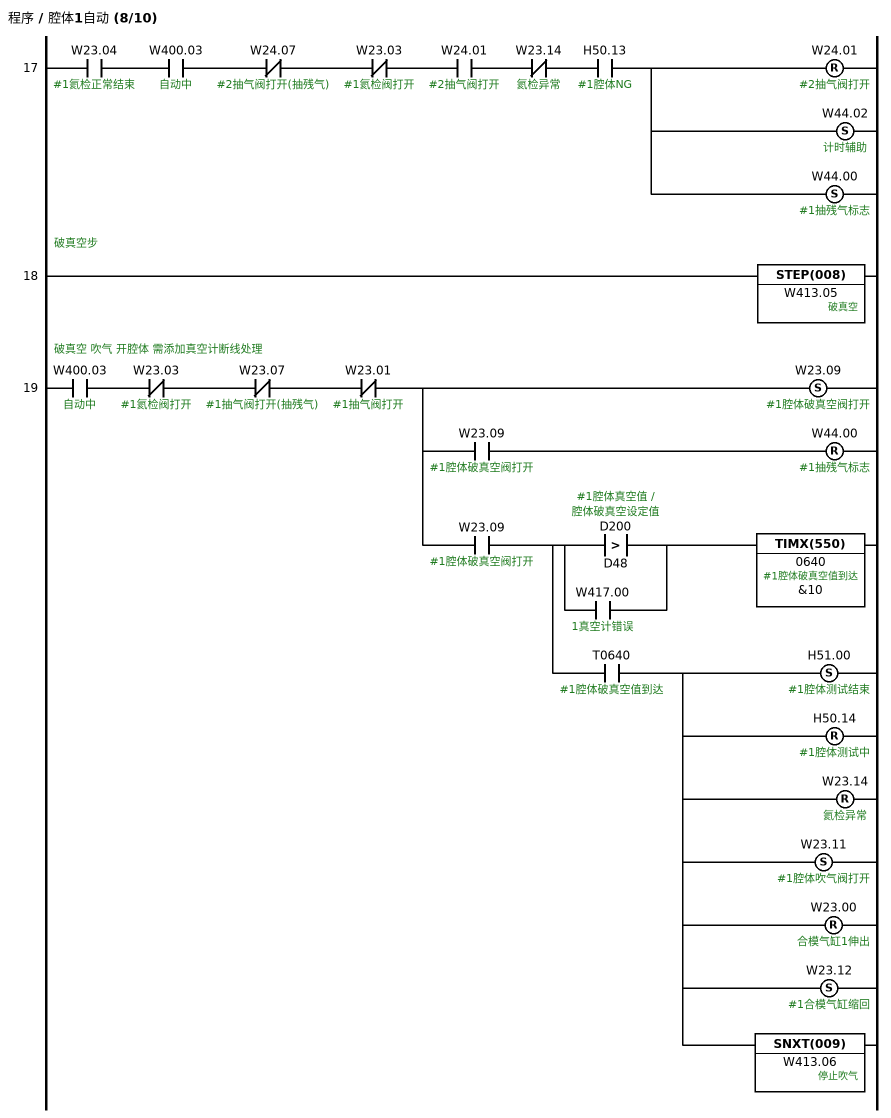
; rung 17
LD W23.04  ; #1氦检正常结束
AND W400.03  ; 自动中
ANDNOT W24.07  ; #2抽气阀打开(抽残气)
ANDNOT W23.03  ; #1氦检阀打开
AND W24.01  ; #2抽气阀打开
ANDNOT W23.14  ; 氦检异常
AND H50.13  ; #1腔体NG
RSET W24.01  ; #2抽气阀打开
SET W44.02  ; 计时辅助
SET W44.00  ; #1抽残气标志
; rung 18: 破真空步
STEP(008) W413.05  ; 破真空
; rung 19: 破真空 吹气 开腔体 需添加真空计断线处理
LD W400.03  ; 自动中
ANDNOT W23.03  ; #1氦检阀打开
ANDNOT W23.07  ; #1抽气阀打开(抽残气)
ANDNOT W23.01  ; #1抽气阀打开
OUT TR0
SET W23.09  ; #1腔体破真空阀打开
AND W23.09  ; #1腔体破真空阀打开
RSET W44.00  ; #1抽残气标志
LD TR0
AND W23.09  ; #1腔体破真空阀打开
OUT TR0
LD>F(333) D200 D48  ; #1腔体真空值, 腔体破真空设定值
OR W417.00  ; 1真空计错误
ANDLD
TIMX(550) 0640 &10  ; #1腔体破真空值到达
LD TR0
AND T0640  ; #1腔体破真空值到达
SET H51.00  ; #1腔体测试结束
RSET H50.14  ; #1腔体测试中
RSET W23.14  ; 氦检异常
SET W23.11  ; #1腔体吹气阀打开
RSET W23.00  ; 合模气缸1伸出
SET W23.12  ; #1合模气缸缩回
SNXT(009) W413.06  ; 停止吹气

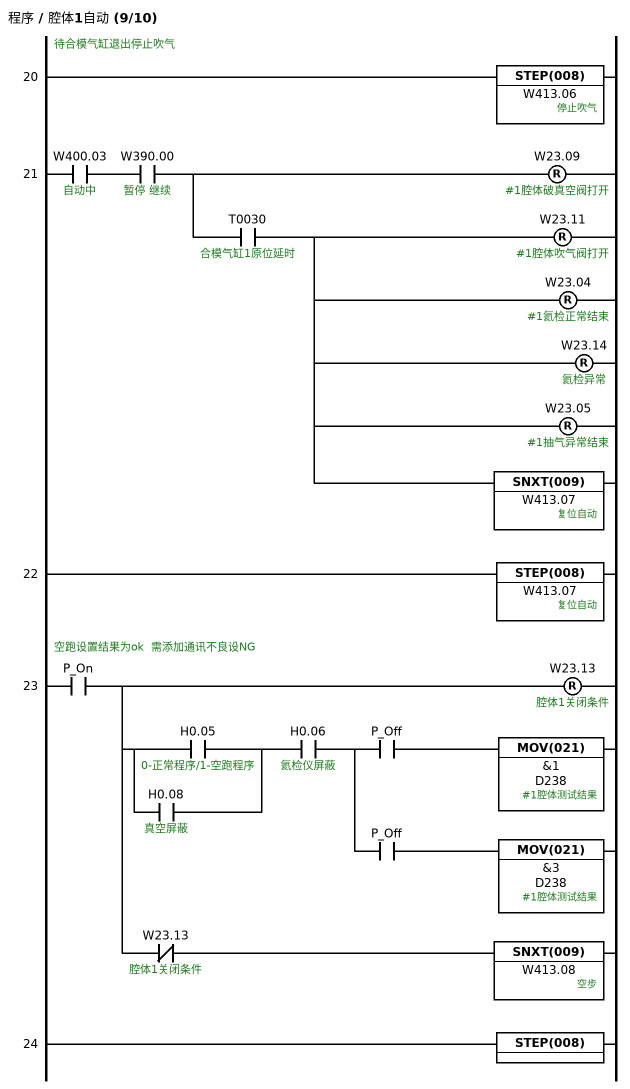
; rung 20: 待合模气缸退出停止吹气
STEP(008) W413.06  ; 停止吹气
; rung 21
LD W400.03  ; 自动中
AND W390.00  ; 暂停 继续
RSET W23.09  ; #1腔体破真空阀打开
AND T0030  ; 合模气缸1原位延时
RSET W23.11  ; #1腔体吹气阀打开
RSET W23.04  ; #1氦检正常结束
RSET W23.14  ; 氦检异常
RSET W23.05  ; #1抽气异常结束
SNXT(009) W413.07  ; 复位自动
; rung 22
STEP(008) W413.07  ; 复位自动
; rung 23: 空跑设置结果为ok  需添加通讯不良设NG
LD P_On
OUT TR0
RSET W23.13  ; 腔体1关闭条件
LD H0.05  ; 0-正常程序/1-空跑程序
OR H0.08  ; 真空屏蔽
ANDLD
AND H0.06  ; 氦检仪屏蔽
OUT TR1
AND P_Off
MOV(021) &1 D238  ; #1腔体测试结果
LD TR1
AND P_Off
MOV(021) &3 D238  ; #1腔体测试结果
LD TR0
ANDNOT W23.13  ; 腔体1关闭条件
SNXT(009) W413.08  ; 空步
; rung 24
STEP(008)

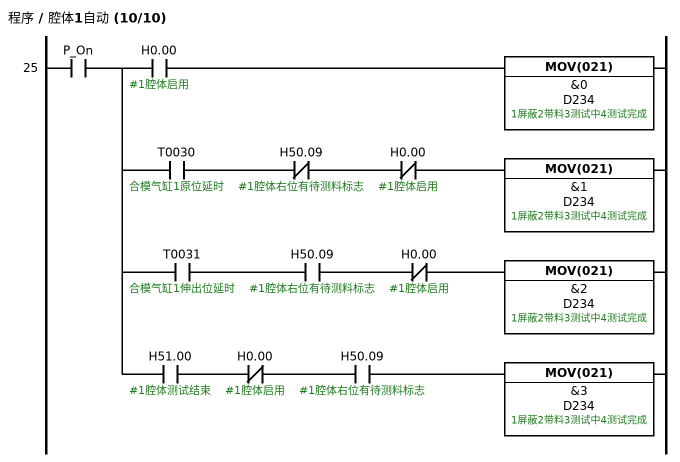
; rung 25
LD P_On
OUT TR0
AND H0.00  ; #1腔体启用
MOV(021) &0 D234  ; 1屏蔽2带料3测试中4测试完成
LD TR0
AND T0030  ; 合模气缸1原位延时
ANDNOT H50.09  ; #1腔体右位有待测料标志
ANDNOT H0.00  ; #1腔体启用
MOV(021) &1 D234  ; 1屏蔽2带料3测试中4测试完成
LD TR0
AND T0031  ; 合模气缸1伸出位延时
AND H50.09  ; #1腔体右位有待测料标志
ANDNOT H0.00  ; #1腔体启用
MOV(021) &2 D234  ; 1屏蔽2带料3测试中4测试完成
LD TR0
AND H51.00  ; #1腔体测试结束
ANDNOT H0.00  ; #1腔体启用
AND H50.09  ; #1腔体右位有待测料标志
MOV(021) &3 D234  ; 1屏蔽2带料3测试中4测试完成

### Section 腔体2自动

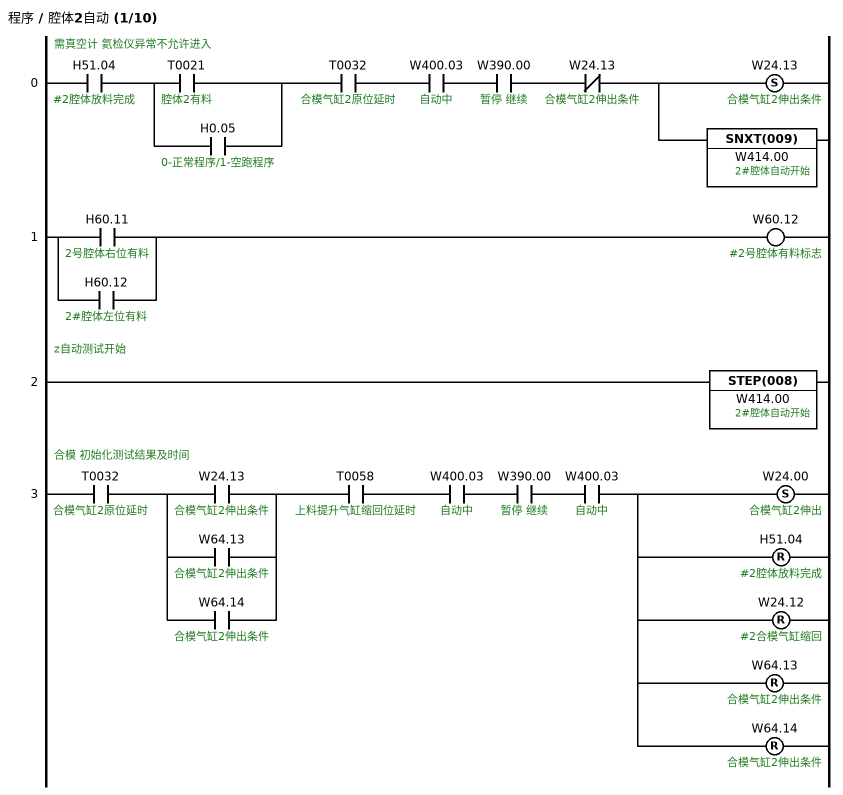
; rung 0: 需真空计 氦检仪异常不允许进入
LD H51.04  ; #2腔体放料完成
LD T0021  ; 腔体2有料
OR H0.05  ; 0-正常程序/1-空跑程序
ANDLD
AND T0032  ; 合模气缸2原位延时
AND W400.03  ; 自动中
AND W390.00  ; 暂停 继续
ANDNOT W24.13  ; 合模气缸2伸出条件
SET W24.13  ; 合模气缸2伸出条件
SNXT(009) W414.00  ; 2#腔体自动开始
; rung 1
LD H60.11  ; 2号腔体右位有料
OR H60.12  ; 2#腔体左位有料
OUT W60.12  ; #2号腔体有料标志
; rung 2: z自动测试开始
STEP(008) W414.00  ; 2#腔体自动开始
; rung 3: 合模 初始化测试结果及时间
LD T0032  ; 合模气缸2原位延时
LD W24.13  ; 合模气缸2伸出条件
OR W64.13  ; 合模气缸2伸出条件
OR W64.14  ; 合模气缸2伸出条件
ANDLD
AND T0058  ; 上料提升气缸缩回位延时
AND W400.03  ; 自动中
AND W390.00  ; 暂停 继续
AND W400.03  ; 自动中
SET W24.00  ; 合模气缸2伸出
RSET H51.04  ; #2腔体放料完成
RSET W24.12  ; #2合模气缸缩回
RSET W64.13  ; 合模气缸2伸出条件
RSET W64.14  ; 合模气缸2伸出条件

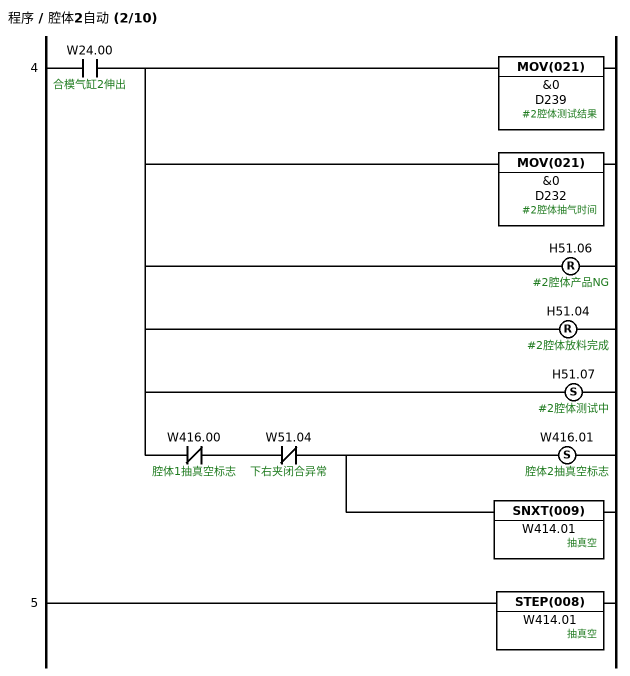
; rung 4
LD W24.00  ; 合模气缸2伸出
MOV(021) &0 D239  ; #2腔体测试结果
MOV(021) &0 D232  ; #2腔体抽气时间
RSET H51.06  ; #2腔体产品NG
RSET H51.04  ; #2腔体放料完成
SET H51.07  ; #2腔体测试中
ANDNOT W416.00  ; 腔体1抽真空标志
ANDNOT W51.04  ; 下右夹闭合异常
SET W416.01  ; 腔体2抽真空标志
SNXT(009) W414.01  ; 抽真空
; rung 5
STEP(008) W414.01  ; 抽真空

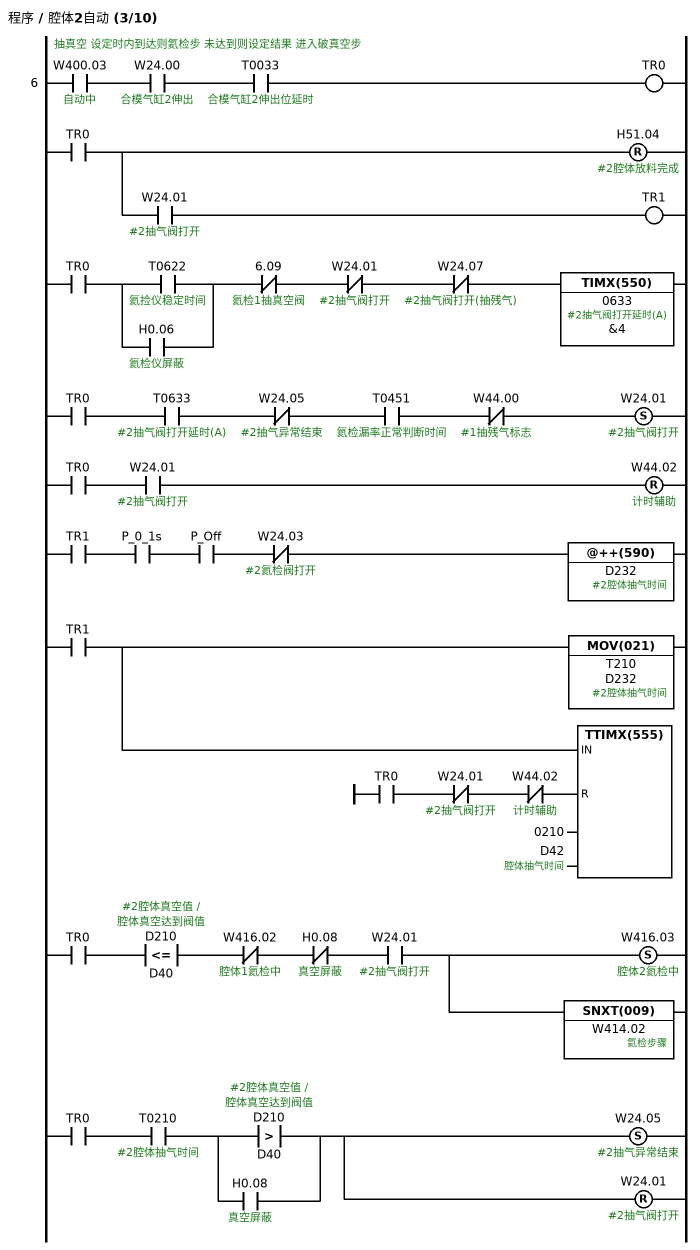
; rung 6: 抽真空 设定时内到达则氦检步 未达到则设定结果 进入破真空步
LD W400.03  ; 自动中
AND W24.00  ; 合模气缸2伸出
AND T0033  ; 合模气缸2伸出位延时
OUT TR0
LD T0622  ; 氦捡仪稳定时间
OR H0.06  ; 氦检仪屏蔽
ANDLD
ANDNOT 6.09  ; 氦检1抽真空阀
ANDNOT W24.01  ; #2抽气阀打开
ANDNOT W24.07  ; #2抽气阀打开(抽残气)
TIMX(550) 0633 &4  ; #2抽气阀打开延时(A)
LD TR0
AND T0633  ; #2抽气阀打开延时(A)
ANDNOT W24.05  ; #2抽气异常结束
AND T0451  ; 氦检漏率正常判断时间
ANDNOT W44.00  ; #1抽残气标志
SET W24.01  ; #2抽气阀打开
LD TR0
AND W24.01  ; #2抽气阀打开
RSET W44.02  ; 计时辅助
LD TR0
RSET H51.04  ; #2腔体放料完成
AND W24.01  ; #2抽气阀打开
OUT TR1
AND P_0_1s
AND P_Off
ANDNOT W24.03  ; #2氦检阀打开
@++(590) D232  ; #2腔体抽气时间
LD TR1
MOV(021) T210 D232  ; #2腔体抽气时间
LD TR0
ANDNOT W24.01  ; #2抽气阀打开
ANDNOT W44.02  ; 计时辅助
TTIMX(555) 0210 D42  ; 腔体抽气时间, #2腔体抽气时间
LD TR0
AND<=F(332) D210 D40  ; #2腔体真空值, 腔体真空达到阀值
ANDNOT W416.02  ; 腔体1氦检中
ANDNOT H0.08  ; 真空屏蔽
AND W24.01  ; #2抽气阀打开
SET W416.03  ; 腔体2氦检中
SNXT(009) W414.02  ; 氦检步骤
LD TR0
AND T0210  ; #2腔体抽气时间
LD>F(333) D210 D40  ; #2腔体真空值, 腔体真空达到阀值
OR H0.08  ; 真空屏蔽
ANDLD
SET W24.05  ; #2抽气异常结束
RSET W24.01  ; #2抽气阀打开

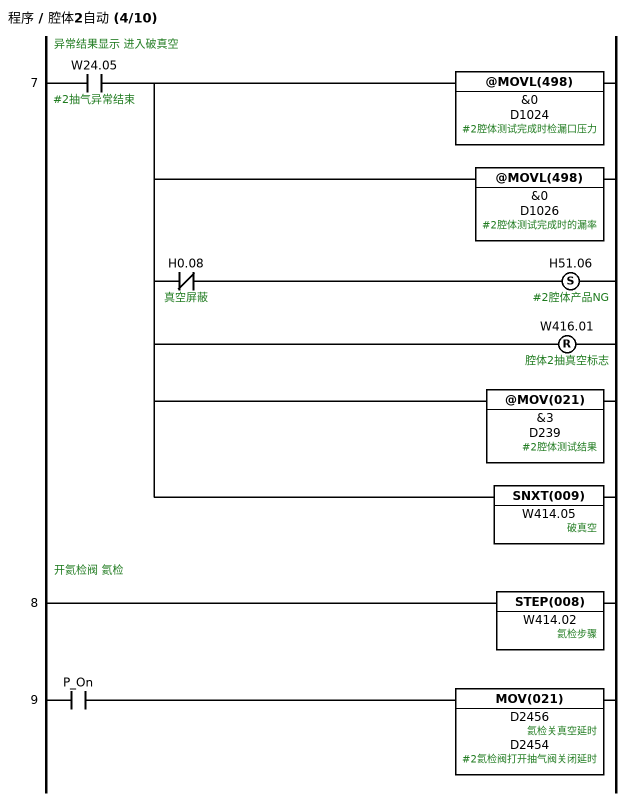
; rung 7: 异常结果显示 进入破真空
LD W24.05  ; #2抽气异常结束
OUT TR0
@MOVL(498) &0 D1024  ; #2腔体测试完成时检漏口压力
@MOVL(498) &0 D1026  ; #2腔体测试完成时的漏率
ANDNOT H0.08  ; 真空屏蔽
SET H51.06  ; #2腔体产品NG
LD TR0
RSET W416.01  ; 腔体2抽真空标志
@MOV(021) &3 D239  ; #2腔体测试结果
SNXT(009) W414.05  ; 破真空
; rung 8: 开氦检阀 氦检
STEP(008) W414.02  ; 氦检步骤
; rung 9
LD P_On
MOV(021) D2456 D2454  ; 氦检关真空延时, #2氦检阀打开抽气阀关闭延时

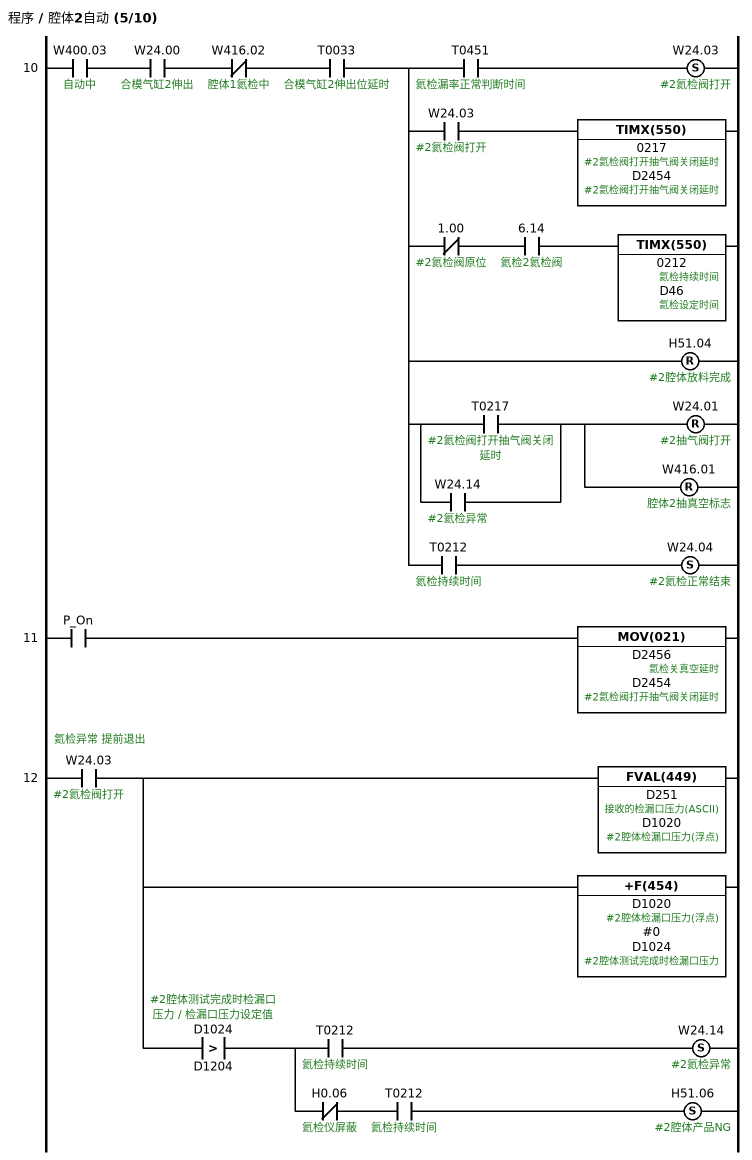
; rung 10
LD W400.03  ; 自动中
AND W24.00  ; 合模气缸2伸出
ANDNOT W416.02  ; 腔体1氦检中
AND T0033  ; 合模气缸2伸出位延时
OUT TR0
AND T0451  ; 氦检漏率正常判断时间
SET W24.03  ; #2氦检阀打开
LD TR0
AND W24.03  ; #2氦检阀打开
TIMX(550) 0217 D2454  ; #2氦检阀打开抽气阀关闭延时
LD TR0
ANDNOT 1.00  ; #2氦检阀原位
AND 6.14  ; 氦检2氦检阀
TIMX(550) 0212 D46  ; 氦检设定时间, 氦检持续时间
LD TR0
RSET H51.04  ; #2腔体放料完成
LD T0217  ; #2氦检阀打开抽气阀关闭延时
OR W24.14  ; #2氦检异常
ANDLD
RSET W24.01  ; #2抽气阀打开
RSET W416.01  ; 腔体2抽真空标志
LD TR0
AND T0212  ; 氦检持续时间
SET W24.04  ; #2氦检正常结束
; rung 11
LD P_On
MOV(021) D2456 D2454  ; 氦检关真空延时, #2氦检阀打开抽气阀关闭延时
; rung 12: 氦检异常 提前退出
LD W24.03  ; #2氦检阀打开
FVAL(449) D251 D1020  ; 接收的检漏口压力(ASCII), #2腔体检漏口压力(浮点)
+F(454) D1020 #0 D1024  ; #2腔体检漏口压力(浮点), #2腔体测试完成时检漏口压力
AND>F(333) D1024 D1204  ; #2腔体测试完成时检漏口压力, 检漏口压力设定值
OUT TR0
AND T0212  ; 氦检持续时间
SET W24.14  ; #2氦检异常
LD TR0
ANDNOT H0.06  ; 氦检仪屏蔽
AND T0212  ; 氦检持续时间
SET H51.06  ; #2腔体产品NG

